{attribute 'analysis' := '-33'}
PROGRAM PRG_UnitTests

VAR
{IF defined (UNIT_TEST)}	
	fbF_RpcSymbolTests_SUT	: FB_F_RpcSymbol_Tests;
	fbRpcTests				: FB_RPC_Tests;
{END_IF}
END_VAR

{IF defined (UNIT_TEST)}

TcUnit.RUN();

{END_IF}

END_PROGRAM

(* stored: Version 1.1.0.1, ProductVersion 3.1.4024.12
   POU PRG_UnitTests: Id {e25ec562-542b-45d4-af41-3a64fbc21fb4}, SpecialFunc None *)
